(* IEC 61131-3 sources: StPos/, 4 files *)

(* ---- StPos.typ ---- *)
(******************************************************************************
 * File: StPos.typ
 * Author: Tyler Matijevich
 * Date: 2021-05-22
*******************************************************************************)

TYPE
	SuperTrakPositionErrorEnum :
		( (*StPos results*)
		stPOS_ERROR_NONE := 0, (*Function call successful*)
		stPOS_ERROR_SERVCHAN := 10, (*The service channel read request returned an error. See SuperTrak library for error code descriptions.*)
		stPOS_ERROR_SECTIONCOUNT, (*SuperTrak section count exceeds the maximum*)
		stPOS_ERROR_SECTIONADDRESS, (*SuperTrak section address exceeds the layout section count*)
		stPOS_ERROR_SECTIONTYPE, (*Invalid SuperTrak section type*)
		stPOS_ERROR_HEADSECTION, (*Invalid head section 1..64*)
		stPOS_ERROR_FLOWDIRECTION, (*Invalid flow direction 0..1*)
		stPOS_ERROR_NETWORKORDER := 100, (*Unexpected SuperTrak section network order*)
		stPOS_ERROR_INPUTORIGIN, (*Invalid input origin section for the given layout section count*)
		stPOS_ERROR_INPUTSECTION, (*Invalid input section for the given layout section count*)
		stPOS_ERROR_INPUTSECTIONPOS, (*Input position exceeds the allowed section position limit*)
		stPOS_ERROR_INPUTGLOBALPOS, (*Input global position exceeds the layout total length limit*)
		stPOS_ERROR_NETWORKGLOBAL (*The global position was not found in the SuperTrak section network*)
		);
	SuperTrakPositionInfoType : 	STRUCT  (*StPos diagnostic information*)
		serviceChannelResult : UINT; (*Service channel read result*)
		serviceChannelParameter : UINT; (*Service channel read parameter associated with serviceChannelResult*)
		section : UINT; (*User address of the section in context of an error*)
		sectionCount : UINT; (*Section count of the system layout*)
		sectionCountMax : UINT; (*Maximum sections allowed in a SuperTrak layout*)
		sectionType : UINT; (*Section type result*)
		sectionTypeMax : UINT; (*Maximum allowed section type*)
		networkIndex : UINT; (*Index in the network layout array of section user addresses*)
		headSection : UINT; (*(Par 1104) Active logical head section *)
		flowDirection : UINT; (*(Par 1105) Active pallet flow direction 0..1*)
		originSection : USINT; (*Input origin section when in context of an error*)
		sectionPosition : DINT; (*Input section position when in context of an error*)
		sectionPositionMax : DINT; (*Maximum allowed input position depending on the section type*)
		globalPosition : DINT; (*Input global position when in context of an error*)
		totalLength : DINT; (*Total length of the valid SuperTrak layout*)
	END_STRUCT;
	SuperTrakSystemLayoutType : 	STRUCT  (*StPos system layout information*)
		sectionCount : USINT; (*Number of sections in the layout*)
		sectionType : ARRAY[0..stPOS_SECTION_MAX]OF USINT; (*Section type, see SuperTrakReadyLayout comments*)
		networkOrder : ARRAY[0..stPOS_SECTION_INDEX]OF USINT; (*Section numbers from left network tail to right network tail*)
		networkMapping : ARRAY[0..stPOS_SECTION_MAX]OF USINT; (*Map from section number 1..64 to network index 0..63*)
		flowOrder : ARRAY[0..stPOS_SECTION_INDEX]OF USINT; (*Section numbers starting at head and continuing in flow direction*)
		layoutLinear : BOOL; (*True - linear, False - loop*)
	END_STRUCT;
END_TYPE

(* ---- Types.typ ---- *)
TYPE
	SuperTrakPositionErrorEnum :
		( (*StPos function call results*)
		stPOS_ERROR_NONE, (*Function call successful*)
		stPOS_ERROR_SERV_CHAN, (*The service channel read request returned an error. See SuperTrak library for error code descriptions.*)
		stPOS_ERROR_LAYOUT, (*Unexpected system layout. Section count or section number out of range.*)
		stPOS_ERROR_SECTION, (*Input section out of range. 1..sectionCount.*)
		stPOS_ERROR_POSITION, (*Input position out of range. 0..1000000 or 0..1030000 for curves.*)
		stPOS_ERROR_ORIGIN (*Input origin section out of range. 1..sectionCount.*)
		);
	SuperTrakPositionDiagType : 	STRUCT  (*StPos position transformation diagnostic information*)
		ServiceChannelResult_1080 : UINT; (*Service channel read result for parameter 1080 - Section Count [UInt16]*)
		ServiceChannelResult_1081 : UINT; (*Service channel read result for parameter 1081 - Section User Address [UInt16]*)
		ServiceChannelResult_1082 : UINT; (*Service channel read result for parameter 1082 - Section Type [UInt16]*)
		SectionCount : UINT; (*Section count of the system layout. 0 if no error.*)
		SectionAddress : UINT; (*Section address index on the system network. 0 if no error.*)
		SectionNumber : UINT; (*Section number at the network address index. 0 if no error.*)
	END_STRUCT;
END_TYPE

(* ---- StPos.fun ---- *)
(******************************************************************************
 * File: StPos.fun
 * Author: Tyler Matijevich
 * Date: 2021-05-22
*******************************************************************************)

FUNCTION SuperTrakGlobalPosition : DINT (*Global position on SuperTrak*)
	VAR_INPUT
		section : USINT; (*Section number*)
		sectionPosition : DINT; (*[um] Position referenced to section's left edge*)
		originSection : USINT; (*First section in layout for global reference*)
		direction : DINT; (*Global direction (Left - 0, Right - 1)*)
		globalPosition : REFERENCE TO DINT; (*[um] Global position result*)
		info : SuperTrakPositionInfoType; (*Diagnostic information*)
	END_VAR
END_FUNCTION

FUNCTION SuperTrakSectionPosition : DINT (*Section position on SuperTrak*)
	VAR_INPUT
		globalPosition : DINT; (*[um] Global position referenced to origin section*)
		originSection : USINT; (*First section in layout for global reference*)
		direction : DINT; (*Global direction (Left - 0, Right - 1)*)
		section : REFERENCE TO USINT; (*Section number result*)
		sectionPosition : REFERENCE TO DINT; (*[um] Section position result referenced to section's left edge*)
		info : SuperTrakPositionInfoType; (*Diagnostic information*)
	END_VAR
END_FUNCTION

FUNCTION SuperTrakTotalLength : DINT (*Total pallet travel length of the SuperTrak section network*)
	VAR_INPUT
		length : REFERENCE TO DINT; (*Pointer to DINT to store the SuperTrak total length*)
		info : SuperTrakPositionInfoType; (*Diagnostic information*)
	END_VAR
END_FUNCTION

FUNCTION SuperTrakSystemLayout : DINT (*SuperTrak system layout*)
	VAR_INPUT
		layout : SuperTrakSystemLayoutType; (*Reference to the system layout structure*)
		info : SuperTrakPositionInfoType; (*Diagnostic information*)
	END_VAR
END_FUNCTION

FUNCTION SuperTrakRefreshLayout : DINT (*Force re-read of SuperTrak system layout after encoder calibration*)
END_FUNCTION

(* ---- StPos.var ---- *)
(******************************************************************************
 * File: StPos.var
 * Author: Tyler Matijevich
 * Date: 2021-05-22
*******************************************************************************)

VAR CONSTANT
	stPOS_SECTION_MAX : USINT := 64; (*Maximum number of sections*)
	stPOS_SECTION_INDEX : USINT := stPOS_SECTION_MAX - 1; (*Size section arrays*)
END_VAR
